SUBAPPLICATION mapping_Uebung_032 (* LED Strip Blinkende LED *)
  (* Standard: 61499-2; Description: Copyright (c) 2023 Meisterschulen am Ostbahnhof This program and the accompanying materials are made available under the terms of the Eclipse Public License 2.0 which is available at https://www.eclipse.org/legal/epl-2.0/ SPDX-License-Identifier: EPL-2.0 *)
  (* Version 1.0, 2023-10-23, Franz Höpfinger, Meisterschulen am Ostbahnhof *)
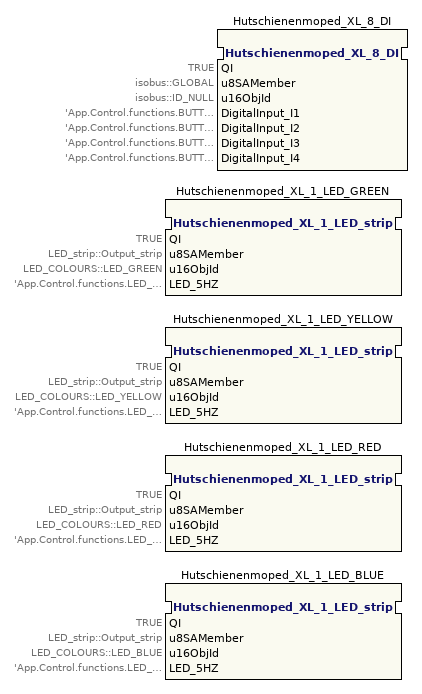
  FBS
    Hutschienenmoped_XL_8_DI : Hutschienenmoped_XL_8_DI(QI := TRUE, u8SAMember := isobus::GLOBAL, u16ObjId := isobus::ID_NULL, DigitalInput_I1 := 'App.Control.functions.BUTTON_GREEN', DigitalInput_I2 := 'App.Control.functions.BUTTON_YELLOW', DigitalInput_I3 := 'App.Control.functions.BUTTON_RED', DigitalInput_I4 := 'App.Control.functions.BUTTON_BLUE');
    Hutschienenmoped_XL_1_LED_YELLOW : Hutschienenmoped_XL_1_LED_strip(QI := TRUE, u8SAMember := LED_strip::Output_strip, u16ObjId := LED_COLOURS::LED_YELLOW, LED_5HZ := 'App.Control.functions.LED_YELLOW_5HZ');
    Hutschienenmoped_XL_1_LED_GREEN : Hutschienenmoped_XL_1_LED_strip(QI := TRUE, u8SAMember := LED_strip::Output_strip, u16ObjId := LED_COLOURS::LED_GREEN, LED_5HZ := 'App.Control.functions.LED_GREEN_5HZ');
    Hutschienenmoped_XL_1_LED_RED : Hutschienenmoped_XL_1_LED_strip(QI := TRUE, u8SAMember := LED_strip::Output_strip, u16ObjId := LED_COLOURS::LED_RED, LED_5HZ := 'App.Control.functions.LED_RED_5HZ');
    Hutschienenmoped_XL_1_LED_BLUE : Hutschienenmoped_XL_1_LED_strip(QI := TRUE, u8SAMember := LED_strip::Output_strip, u16ObjId := LED_COLOURS::LED_BLUE, LED_5HZ := 'App.Control.functions.LED_BLUE_5HZ');
  END_FBS
END_SUBAPPLICATION
